FUNCTION_BLOCK ChunkedRequestData_TestSuite EXTENDS TcUnit.FB_TestSuite
VAR
END_VAR

TestChunkedPayloadStoredCorrectly_10Chunks();
TestChunkedPayloadStoredCorrectly_2Chunks();
TestCorrectPayloadSizeInBytes_20Bytes();
TestCorrectPayloadSizeInBytes_100Bytes();
TestIsCompleteOnceAllChunksAdded();
TestTryAddChunkedPayloadReturnsFalseWhenTooBig();
TestTryAddChunkedPayloadReturnsTrueWhenValid();

METHOD TestChunkedPayloadStoredCorrectly_10Chunks
VAR
	chunkedRequestData : ChunkedRequestSessionData(3,10); // results in 30 bytes
	dataChunk1 : STRING(2) := 'ab'; // results in 3 bytes
	dataChunk2 : STRING(2) := 'cd'; // results in 3 bytes
	dataChunk3 : STRING(2) := 'ef'; // results in 3 bytes
	dataChunk4 : STRING(2) := 'gh'; // results in 3 bytes
	dataChunk5 : STRING(2) := 'ij'; // results in 3 bytes
	dataChunk6 : STRING(2) := 'kl'; // results in 3 bytes
	dataChunk7 : STRING(2) := 'mn'; // results in 3 bytes
	dataChunk8 : STRING(2) := 'op'; // results in 3 bytes
	dataChunk9 : STRING(2) := 'qr'; // results in 3 bytes
	dataChunk10 : STRING(2) := 'st'; // results in 3 bytes
	dataAddress : PVOID;
	dataSize : UDINT;
	result : STRING(29);
	expected : STRING(29) := 'abcdefghijklmnopqrst'; // results in 30 bytes
END_VAR
TEST('TestChunkedPayloadStoredCorrectly_10Chunks');

memset(ADR(result),0,SIZEOF(result));

chunkedRequestData.TryAddChunkedPayload(ADR(dataChunk1), SIZEOF(dataChunk1), 1);
chunkedRequestData.TryAddChunkedPayload(ADR(dataChunk2), SIZEOF(dataChunk2), 2);
chunkedRequestData.TryAddChunkedPayload(ADR(dataChunk3), SIZEOF(dataChunk3), 3);
chunkedRequestData.TryAddChunkedPayload(ADR(dataChunk4), SIZEOF(dataChunk4), 4);
chunkedRequestData.TryAddChunkedPayload(ADR(dataChunk5), SIZEOF(dataChunk5), 5);
chunkedRequestData.TryAddChunkedPayload(ADR(dataChunk6), SIZEOF(dataChunk6), 6);
chunkedRequestData.TryAddChunkedPayload(ADR(dataChunk7), SIZEOF(dataChunk7), 7);
chunkedRequestData.TryAddChunkedPayload(ADR(dataChunk8), SIZEOF(dataChunk8), 8);
chunkedRequestData.TryAddChunkedPayload(ADR(dataChunk9), SIZEOF(dataChunk9), 9);
chunkedRequestData.TryAddChunkedPayload(ADR(dataChunk10), SIZEOF(dataChunk10), 10);

dataAddress := chunkedRequestData.PayloadAddress;
dataSize := chunkedRequestData.PayloadSizeInBytes;

memcpy(ADR(result),dataAddress,dataSize);

AssertEquals(
	Expected := expected,
	Actual := result,
	Message := 'Did not correctly assemble the chunked string data'
);

TEST_FINISHED();
END_METHOD

METHOD TestChunkedPayloadStoredCorrectly_2Chunks
VAR
	chunkedRequestData : ChunkedRequestSessionData(4,2); // results in 8 bytes
	dataChunk1 : STRING(3) := 'foo'; // results in 4 bytes
	dataChunk2 : STRING(3) := 'bar'; // results in 4 bytes
	dataAddress : PVOID;
	dataSize : UDINT;
	result : STRING(7);
	expected : STRING(7) := 'foobar'; // results in 8 bytes
END_VAR
TEST('TestChunkedPayloadStoredCorrectly_2Chunks');

memset(ADR(result),0,SIZEOF(result));

chunkedRequestData.TryAddChunkedPayload(ADR(dataChunk1), SIZEOF(dataChunk1), 1);
chunkedRequestData.TryAddChunkedPayload(ADR(dataChunk2), SIZEOF(dataChunk2), 2);

dataAddress := chunkedRequestData.PayloadAddress;
dataSize := chunkedRequestData.PayloadSizeInBytes;

memcpy(ADR(result),dataAddress,dataSize);

AssertEquals(
	Expected := expected,
	Actual := result,
	Message := 'Did not correctly assemble the chunked string data'
);

TEST_FINISHED();
END_METHOD

METHOD TestCorrectPayloadSizeInBytes_100Bytes
VAR
	chunkedRequestData : ChunkedRequestSessionData(20,5);
	result : UDINT;
	expected : UDINT := 100;
END_VAR
TEST('TestCorrectPayloadSizeInBytes_100Bytes');

result := chunkedRequestData.PayloadSizeInBytes;

AssertEquals(
	Expected := expected,
	Actual := result,
	Message := 'Did not create the correct payload size based on the constructor arguments'
);

TEST_FINISHED();
END_METHOD

METHOD TestCorrectPayloadSizeInBytes_20Bytes
VAR
	chunkedRequestData : ChunkedRequestSessionData(2,10);
	result : UDINT;
	expected : UDINT := 20;
END_VAR
TEST('TestCorrectPayloadSizeInBytes_20Bytes');

result := chunkedRequestData.PayloadSizeInBytes;

AssertEquals(
	Expected := expected,
	Actual := result,
	Message := 'Did not create the correct payload size based on the constructor arguments'
);

TEST_FINISHED();
END_METHOD

METHOD TestIsCompleteOnceAllChunksAdded
VAR
	chunkedRequestData : ChunkedRequestSessionData(4,2);
	dataChunk1 : STRING(3) := 'foo';
	dataChunk2 : STRING(3) := 'bar';
	isComplete : BOOL;
END_VAR
TEST('TestIsCompleteOnceAllChunksAdded');

isComplete := chunkedRequestData.IsComplete;

AssertFalse(
	Condition := isComplete,
	Message := 'Incorrectly reported as IsComplete with 0/2 chunks added'
);

chunkedRequestData.TryAddChunkedPayload(ADR(dataChunk1), SIZEOF(dataChunk1), 1);
isComplete := chunkedRequestData.IsComplete;

AssertFalse(
	Condition := isComplete,
	Message := 'Incorrectly reported as IsComplete with 1/2 chunks added'
);

chunkedRequestData.TryAddChunkedPayload(ADR(dataChunk2), SIZEOF(dataChunk2), 2);
isComplete := chunkedRequestData.IsComplete;

AssertTrue(
	Condition := isComplete,
	Message := 'Failed to reported IsComplete with 2/2 chunks added'
);

TEST_FINISHED();
END_METHOD

METHOD TestTryAddChunkedPayloadReturnsFalseWhenTooBig
VAR
	chunkedRequestData : ChunkedRequestSessionData(4,1);
	dataChunk : STRING(10) := 'foo';
	added : BOOL;
END_VAR
TEST('TestTryAddChunkedPayloadReturnsFalseWhenTooBig');

added := chunkedRequestData.TryAddChunkedPayload(ADR(dataChunk), SIZEOF(dataChunk), 1);

AssertFalse(
	Condition := added,
	Message := 'Incorrectly reported that the try was successful'
);

TEST_FINISHED();
END_METHOD

METHOD TestTryAddChunkedPayloadReturnsTrueWhenValid
VAR
	chunkedRequestData : ChunkedRequestSessionData(4,1);
	dataChunk : STRING(3) := 'foo';
	added : BOOL;
END_VAR
TEST('TestTryAddChunkedPayloadReturnsTrueWhenValid');

added := chunkedRequestData.TryAddChunkedPayload(ADR(dataChunk), SIZEOF(dataChunk), 1);

AssertTrue(
	Condition := added,
	Message := 'Incorrectly reported that the try failed'
);

TEST_FINISHED();
END_METHOD

END_FUNCTION_BLOCK

(* stored: Version 1.1.0.1, ProductVersion 3.1.4024.12
   POU ChunkedRequestData_TestSuite: Id {a81a4899-70aa-4d46-a8f0-d0593f416472}, SpecialFunc None
   Method TestChunkedPayloadStoredCorrectly_10Chunks: Id {216291d5-8830-40d3-96a5-04ab61b10e06}
   Method TestChunkedPayloadStoredCorrectly_2Chunks: Id {7c47ebe3-8d1b-4014-8d3e-967c884e9f47}
   Method TestCorrectPayloadSizeInBytes_100Bytes: Id {12e658ae-8be5-4bd8-b0c0-a9c774b6c472}
   Method TestCorrectPayloadSizeInBytes_20Bytes: Id {312b4172-8a90-419a-9115-ccbe4031c356}
   Method TestIsCompleteOnceAllChunksAdded: Id {ad28390d-dfaa-4495-b441-2f3c8b567e33}
   Method TestTryAddChunkedPayloadReturnsFalseWhenTooBig: Id {268bd65c-853e-45ae-be79-d89a47f97f0e}
   Method TestTryAddChunkedPayloadReturnsTrueWhenValid: Id {9a498d20-6c9a-4d02-89a0-d08117d9f4e5} *)
